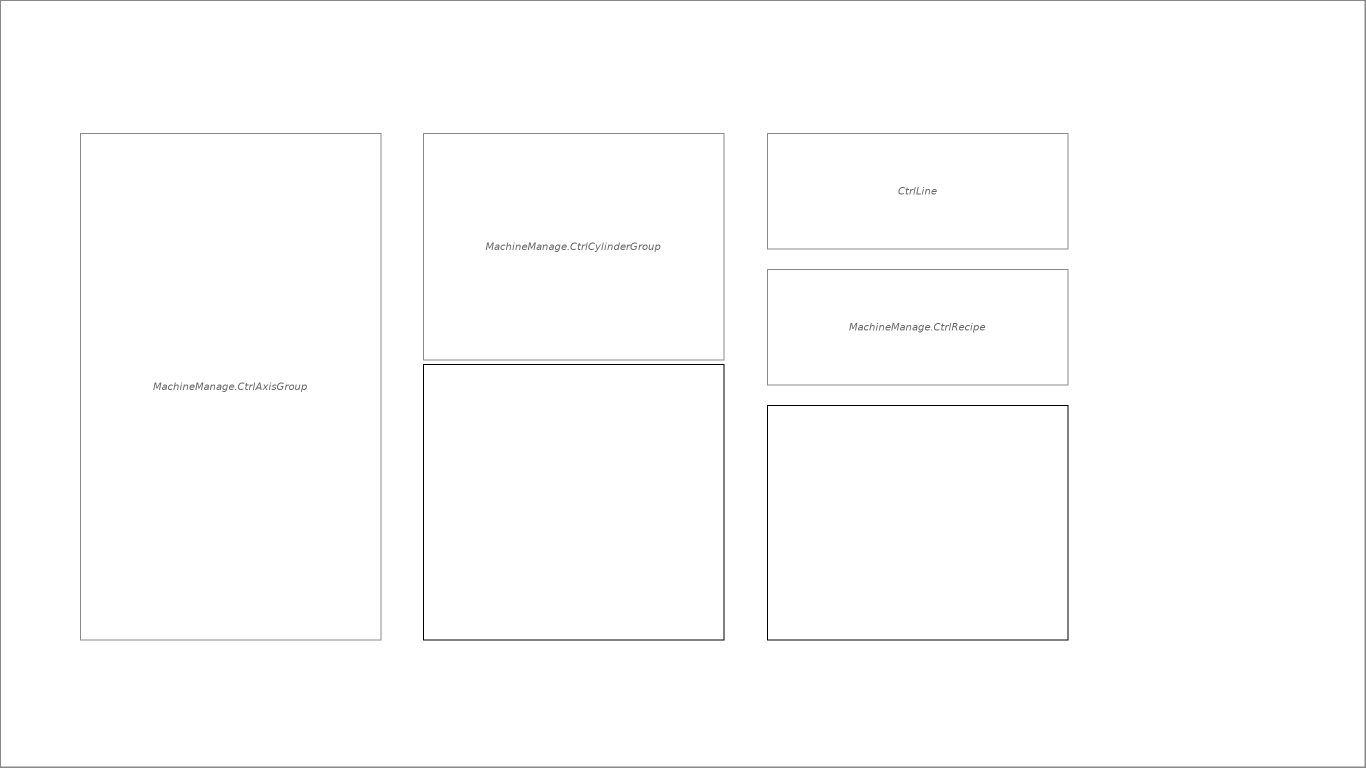
VISUALIZATION PageSetting  // 1366x768
    Frame (0,0 1366x768)
        shows FrameMain()
    Frame (80,133 301x507)
        shows MachineManage.CtrlAxisGroup(System := G_stSystem, Axis := G_arrAxis, Data := G_arrAxisData)
    Frame (423,133 301x227)
        shows MachineManage.CtrlCylinderGroup(System := G_stSystem, Cylinder := G_arrCylinder, CylinderData := G_arrCylinderData)
    RoundedRectangle (767,405 301x235), text list: 'ManualText', text index: 0
    Frame (767,269 301x116)
        shows MachineManage.CtrlRecipe()
    Frame (767,133 301x116)
        shows CtrlLine()
    RoundedRectangle (423,364 301x276), text list: 'ManualText', text index: 1
END_VISUALIZATION

(* stored: Version 1.1.0.1, ProductVersion 3.1.4024.3
   Visu PageSetting: Id {7058b3c2-e93a-4397-ac33-1724fc29a018} *)
